FUNCTION_BLOCK FB_PumpController
VAR_INPUT
	nTargetPressure : USINT := 9; // Volts
	nMaximumPressure : USINT := 10;
	nMinimumPressure : USINT := 8;
	nInitialPressure : REAL;
END_VAR
VAR_OUTPUT
	bPumpState : BOOL := FALSE;
END_VAR
VAR
	nPumpHysteresis : REAL := 0.25;
	nLeakHysteresis : REAL := 0.5;
	nPrevPressure : REAL := nInitialPressure;
	bCheckedForLeak : BOOL := FALSE;
	
	// After <nPumpPollDelay> consecutive increases from pump, check if it's 
	// increased by at least <nPumpBrokenHysteresis>,
	nBrokenPumpHysteresis : REAL := 0.2;
	nBrokenPrevPressure : REAL := nInitialPressure;
	nPumpPollDelay : UINT := 50;
	nPollCount : UINT := 0;

END_VAR

METHOD PRIVATE LeakDetection : BOOL
VAR
	nPressureDiff : REAL;
END_VAR
IF bCheckedForLeak THEN
	nPressureDiff := nPrevPressure - GVL_VAR.nPressure;
	nPollCount := nPollCount + 1;
	IF nPressureDiff > nLeakHysteresis THEN
		GVL_VAR.bLeakDetected := TRUE;
	ELSIF nPollCount > nPumpPollDelay-1 THEN
		nPressureDiff := GVL_VAR.nPressure - nBrokenPrevPressure;
		IF nPressureDiff < nBrokenPumpHysteresis THEN
			GVL_VAR.bBrokenPump := TRUE;
		END_IF
		nBrokenPrevPressure := GVL_VAR.nPressure;
		nPollCount := 0;
	ELSE
		GVL_VAR.bLeakDetected := FALSE;
	END_IF
	nPrevPressure := GVL_VAR.nPressure;
ELSE
	nPrevPressure := GVL_VAR.nPressure;
	nBrokenPrevPressure := GVL_VAR.nPressure;
	bCheckedForLeak := TRUE;
	nPollCount := 1;
END_IF
END_METHOD

METHOD ResetLeakCheck : BOOL
bCheckedForLeak := FALSE;
nPollCount := 0;
ResetLeakCheck := TRUE;
END_METHOD

METHOD Run
VAR_INPUT
	bState : BOOL;
END_VAR
IF bState THEN
	IF GVL_VAR.nPressure < nTargetPressure-nPumpHysteresis OR GVL_VAR.nPressure < nMinimumPressure-nPumpHysteresis THEN
		bPumpState := TRUE;
		LeakDetection();
	ELSIF GVL_VAR.nPressure > nTargetPressure+nPumpHysteresis OR GVL_VAR.nPressure > nMaximumPressure+nPumpHysteresis THEN
		bPumpState := FALSE;
		ResetLeakCheck();
	END_IF
ELSE
	bPumpState := FALSE;
	ResetLeakCheck();
END_IF
END_METHOD

END_FUNCTION_BLOCK

(* stored: Version 1.1.0.1, ProductVersion 3.1.4024.12
   POU FB_PumpController: Id {a50fad6d-a003-4691-b885-4dda779a3353}, SpecialFunc None
   Method LeakDetection: Id {472df253-a6d4-49df-961f-0d688ac52440}
   Method ResetLeakCheck: Id {2a0dfab5-7ee0-416b-89cd-4cbe13014288}
   Method Run: Id {eeca5ea1-f0a1-4ca1-9d59-493b90ef8339} *)
